TYPE E_DataExchangeLD :
(
	IDLE,
	ConnectServer,
	ExchangeData,
	Succeed,
	ERROR
)UDINT;
END_TYPE

(* stored: Version 1.1.0.1, ProductVersion 3.1.4024.11
   DUT E_DataExchangeLD: Id {22af2a7f-2d74-4bd7-98e9-4ca1f9e7646b} *)
